% RSLogix 500 project Encoder 1200BWA.RSS, saved by version 11.00.00.00 %
PROJECT "UNTITLED"    % processor: MicroLogix 1200 %

PROGRAM FILES
  LAD 2   7 rungs
  LAD 3 "HSC"  1 rungs  % Encoder %

DATA FILES
  O0 OUTPUT  4 elements
  I1 INPUT  4 elements
  S2 STATUS  66 elements
  B3 BINARY  1 elements
  T4 TIMER  1 elements
  C5 COUNTER  4 elements
  R6 CONTROL  1 elements
  N7 INTEGER  1 elements
  F8 FLOAT  1 elements
  L9 HSC  3 elements

LADDER 2
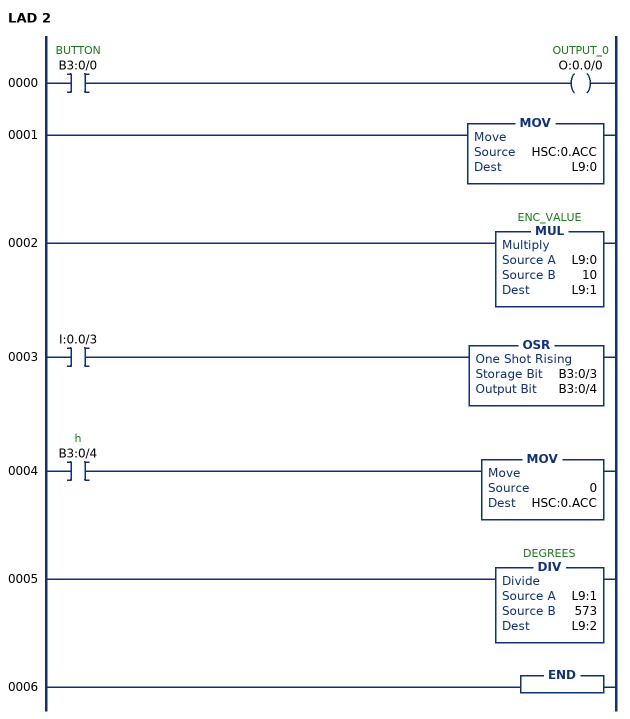
% Rung: 0 %
SOR XIC B3:0/0 OTE O:0.0/0 EOR
%   B3:0/0  BUTTON %
%   O:0.0/0  OUTPUT_0 %
% Rung: 1 %
SOR MOV HSC:0.ACC L9:0 EOR
% Rung: 2 %
SOR MUL L9:0 10 L9:1 EOR
%   L9:1  ENC_VALUE %
% Rung: 3 %
SOR XIC I:0.0/3 OSR B3:0/3 B3:0/4 EOR
%   B3:0/4  "h" %
% Rung: 4 %
SOR XIC B3:0/4 MOV 0 HSC:0.ACC EOR
%   B3:0/4  "h" %
% Rung: 5 %
SOR DIV L9:1 573 L9:2 EOR
%   L9:1  ENC_VALUE %
%   L9:2  DEGREES %
% Rung: 6 %
SOR END EOR

OTHER DOCUMENTED ADDRESSES
  B3:0/1  RES
  B3:0/9  COUNT_DOWN
  C5:0  CLOCK
  HSC:0.5  VALUE
  HSC:0.7  HIGH_SET_POINT
  I:0.0/0  HSC
  I:0.0/4  PHOTO_EYE
  N7:0  PULSES

DATA TABLE (non-zero values as saved)
DATA B3
% B3:0 % 0X0002
DATA C5
% .PRE .ACC %
% C5:0 % 500 0
% C5:1 % 0 -11
DATA N7
% N7:0 % 32767
